ABB RobotStudio station: Station_[09.05.13]3.rsstn

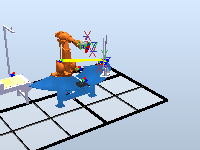
Station Station_[09.05.13] (saved by RobotStudio format 3)
Controller IRB2400_10kg_1.5m_3, task T_ROB1: task frame (RAPID world) sits at (0, 0, 226) mm in the station
Controller IRB2400_10kg_1.5m_3
  mechanical unit ROB_1: IRB2400_10_150__02, 6 joints, base frame (0, 0, -10) mm
Layout (positions relative to the parent item):
  - IRB2400_10_150__02 [mechanism, from Robots\IRB2400_10_150__02.rslib] at (0, 0, 216) mm; joint values [0, 0, 0, 0, 0, 0] (rad or m)
  - Table3_2 [part]
  - SC_RightDispenser [smart component] at (848.89, 660.39, 707) mm, rotated rx 0 ry 0 rz -142.5 deg
      signals: DI diNewPin, DO doPinInPosition2, DO doPinInPosition1
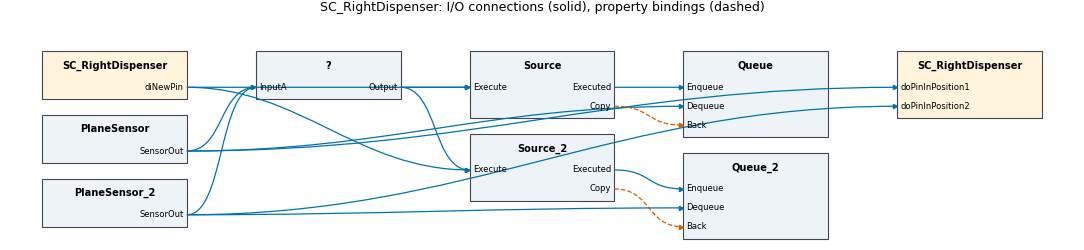
      connections:
        SC_RightDispenser.diNewPin -> Source.Execute
        Source.Executed -> Queue.Enqueue
        PlaneSensor.SensorOut -> Queue.Dequeue
        PlaneSensor.SensorOut -> SC_RightDispenser.doPinInPosition1
        PlaneSensor.SensorOut -> ?.InputA
        ?.Output -> Source.Execute
        SC_RightDispenser.diNewPin -> Source_2.Execute
        Source_2.Executed -> Queue_2.Enqueue
        PlaneSensor_2.SensorOut -> Queue_2.Dequeue
        PlaneSensor_2.SensorOut -> SC_RightDispenser.doPinInPosition2
        PlaneSensor_2.SensorOut -> ?.InputA
        ?.Output -> Source_2.Execute
        Source.Copy => Queue.Back
        Source_2.Copy => Queue_2.Back
    - Dispenser [part]
    - Source [smart component]
        properties: Source=Pin; Copy=(none); Parent=(none); Position=[-0.078 0.0985 0.189]; Orientation=[0 0 0]; Transient=false
        signals: DI Execute, DO Executed
    - Queue [smart component]
        properties: Back=(none); Front=(none); Queue={baa7ba2a-e563-400f-ae00-338ac9d6b310};{166c1fa7-f084-4893-8c68-a7378bc4935a};{0c8467ce-4cb3-4075-8f36-e6447ecc44ba};{a4931bd6-61c0-4022-957d-34420e4f6ad0};{b2f85a70-4d19-413a-b019-3afa180c1445};{512256d1-278f-462d-98f1-9ffcbd4d9afc};{849db594-4dfe-4c58-a8bd-451d21853566};{c968444c-bd1a-4f2f-bbaa-bfd3e7f50be5};{53c4b951-dfc2-4c08-b51d-efe4876241dc};{64f07cc2-7ba3-4255-a888-147bdde81c96};{5e5e12c0-75f5-4fd7-8049-5710cdd06950};{7bc2919c-0f2a-489c-9e4c-df3bff6561ed};{5aa4b278-0833-4ca9-af8d-253aa8523874};{1baac950-fc54-4ea7-852c-7f888843f6f9};{b4b16473-bd2b-40f5-a110-90fbcba822d9};{d003a69b-5307-4c56-b226-d498155ba824};{d659394f-77c7-41ee-9797-cd61472f6401};{a8294731-aa9f-4324-81a7-55ebbef1ff1c};{1eff712e-2c63-4fa8-99b0-fad1482486d3};{b15f9735-19cd-4f7a-8d4f-e540a16427f5};{02485707-3f80-4cc3-94a6-af0fe382acfb};{ec0e8ce0-b480-4ff5-b740-0a7d244ffb35};{21e78636-7eb3-4061-8dde-926c3e464303};{0772fef3-b80e-464b-9cad-322a585d167a};{d8ed8ead-e522-4938-9c7c-7997e1d5aae1};{4dfefca0-2913-4484-9455-684dfc1cbf5a};{f8c8569f-a97f-4f57-84f0-3da59c0f2755};{9fd95979-e5cf-4fa7-b177-2c560699c82c};{84f56170-3294-4345-a728-b2bfe69be833};{b3710d51-6f0f-48ac-9b0f-811ac7c7d083};{c8300349-23e3-4531-beb4-4210900096fb};{31c2e06e-432b-4cd5-8dfd-12cdd0c38bbf};{f6bc1e00-ec05-46bf-9f1a-fcc25cb6084b};{46f4262a-e9c9-45b1-8eff-bed77a1a9e5b};{07cc3b07-c3da-44db-b33b-99881492d9cc};{0c369fdb-a0e7-4beb-a0c1-abd25c6b2a43};{d9cb4cdb-12a7-4146-bf1e-65335fe6fd56};{f09a15e7-f9e4-4c16-add7-657cccb8590f}; NumberOfObjects=0
        signals: DI Enqueue, DI Dequeue, DI Clear, DI Delete, DI DeleteAll
    - LinearMover [smart component]
        properties: Object=Queue; Direction=[0 0 -0.07]; Speed=0.05; Reference=Global; ReferenceObject=(none)
        signals: DI Execute
    - PlaneSensor [smart component]
        properties: Origin=[-0.0530000000000006 0.1235 0.1195]; Axis1=[-0.03 0 0]; Axis2=[0 -0.04 0]; SensedPart=(none)
        signals: DI Active, DO SensorOut
      - _sensorPart_ [part]
    - Pin [part] at (-78, 98.5, 189) mm
    - Source_2 [smart component]
        properties: Source=Pin_2; Copy=(none); Parent=(none); Position=[-0.078 -0.0985 0.198]; Orientation=[0 0 0]; Transient=false
        signals: DI Execute, DO Executed
    - Queue_2 [smart component]
        properties: Back=(none); Front=(none); Queue={1c26a820-5f81-4fc8-b661-270a696b215b};{079caa1e-4b65-4731-ac2d-b38991013e84};{04249497-c8e4-4d2b-8d23-0d0c3b1232f2};{9b46111e-8043-4ec7-820f-f6b1f3216e0a};{190405bf-72c0-4a75-968d-0e05791ba659};{cdaa2867-23d2-4f9c-8306-ddafce1e9ac9};{a0d1b5cc-bcdc-4e7d-b91f-09bc5bc174e5};{802900b3-44c0-4e10-9d61-adfd75a0d86d};{e1828195-6a4a-4e48-b78f-f1287aff9cdc};{27d5d252-1980-452a-aff5-49173c411714};{b44ede4c-8dd3-43ce-8da4-3f1fb091dc7f};{168b000f-829e-439e-a2b5-5bc5735400ce};{aacdfd62-2178-4132-b345-2cd6db76197d};{33bd895a-7dcf-445c-8a77-0a7b01e583dc};{c1a42cbc-38c3-48e5-a615-b149ac9d8780};{fcea76f5-b349-47ef-a520-1d1e9307533b};{d936eec8-07d3-4a18-b33b-be549f4009da};{161ff837-8ce6-447d-8217-59dc5e5add53};{a4db4600-beb4-451b-b75b-f36278185638};{fac26080-080b-42e5-8e31-79509598499f};{631b6ef4-884c-4e99-a73e-a0a20b005bbd};{c6922cb5-858b-4dce-bc49-d50c5bb6ff29};{df2a1232-f236-477f-a341-c0e7247ec374};{648e1593-9b95-4c8f-9a3a-4728290fef8c};{9aba8fcf-9d7f-441d-92fe-144ce1ccaea8}; NumberOfObjects=0
        signals: DI Enqueue, DI Dequeue, DI Clear, DI Delete, DI DeleteAll
    - LinearMover_2 [smart component]
        properties: Object=Queue_2; Direction=[0 0 -0.07]; Speed=0.05; Reference=Global; ReferenceObject=(none)
        signals: DI Execute
    - PlaneSensor_2 [smart component]
        properties: Origin=[-0.053 -0.1235 0.1195]; Axis1=[-0.03 0 0]; Axis2=[0 0.04 0]; SensedPart=(none)
        signals: DI Active, DO SensorOut
      - _sensorPart_ [part]
    - Pin_2 [part] at (-78, -98.5, 189) mm
  - Pallet [part] at (1211.56, -23.95, 701.75) mm, rotated rx 0 ry -0.05 rz -179.99 deg
  - NewSmartGripper[040513] [smart component] at (940, 0, 1671) mm, rotated rx 0 ry 90 rz 0 deg
      signals: DO doPinAttached, DI diAttachPin, DO doPalletAttached, DO doGripperTouchesTable
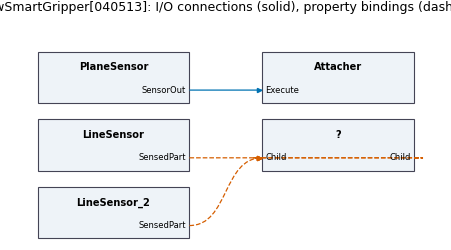
      connections:
        PlaneSensor.SensorOut -> Attacher.Execute
        LineSensor.SensedPart => ?.Child
        ?.Child => ?.Child
        LineSensor_2.SensedPart => ?.Child
        ?.Child => ?.Child
    - LineSensor [smart component, from Components\LineSensor.rslib]
        properties: Start=[0.03 0 0.1702]; End=[0.03 0 0.16]; Radius=0.002; SensedPart=(none); SensedPoint=[0 0 0]
      - _sensorPart_ [part]
    - LineSensor_2 [smart component, from Components\LineSensor.rslib]
        properties: Start=[-0.109 0.07175 0.18]; End=[-0.109 0.07175 0.1]; Radius=0.0012; SensedPart=(none); SensedPoint=[0 0 0]
      - _sensorPart_ [part]
    - LineSensor_3 [smart component, from Components\LineSensor.rslib]
        properties: Start=[-0.142 0 0.04]; End=[-0.12 0 0.04]; Radius=0.004; SensedPart=(none); SensedPoint=[0 0 0]
      - _sensorPart_ [part]
    - PoseMover [smart component, from Components\PoseMover.rslib]
        properties: Mechanism=NewGripperMech; Pose=3; Duration=0.2
    - PoseMover_2 [smart component, from Components\PoseMover.rslib]
        properties: Mechanism=NewGripperMech; Pose=2; Duration=0.2
    - NewGripperMech [mechanism] at (0, 0, 0) mm; joint values [-0.008, 0.008] (rad or m)
        TCP tTine at (-114.5, 0, 234.15) mm, rotated rx 0 ry 0 rz 180 deg
        TCP tGrip at (30, 0, 180) mm, rotated rx 0 ry -90 rz 0 deg
        links: L1, L2, L3
    - LogicGateDetachPin [smart component, from Components\LogicGate.rslib]
        properties: Operator=NOT; Delay=0
    - LogicSRLatchPalletAttached [smart component, from Components\LogicSRLatch.rslib]
    - LogicGateTouchTableANDPallet [smart component, from Components\LogicGate.rslib]
        properties: Operator=AND; Delay=0
    - PlaneSensor [smart component, from Components\PlaneSensor.rslib]
        properties: Origin=[-0.1 -0.05 0.055]; Axis1=[0.02 0 0]; Axis2=[0 0.1 0]; SensedPart=(none)
      - _sensorPart_ [part]
    - LinearMover [smart component, from Components\LinearMover.rslib]
        properties: Object=Pallet; Direction=[0 0 -1]; Speed=0.1; Reference=Object; ReferenceObject=PlaneSensor
    - Positioner [smart component, from Components\Positioner.rslib]
        properties: Object=Pallet; Position=[-0.143 -0.11 0.273]; Orientation=[0 1.5707963267949 0]; Reference=Object; ReferenceObject=PlaneSensor
    - Attacher [smart component, from Components\Attacher.rslib]
        properties: Parent=NewSmartGripper[040513]; Flange=0; Child=Pallet; Mount=false; Offset=[0 0 0]; Orientation=[0 0 0]
    - LinearMover_stop [smart component, from Components\LinearMover.rslib]
        properties: Object=Pallet; Direction=[0 0 1E-07]; Speed=1E-07; Reference=Object; ReferenceObject=PlaneSensor
  - SmartComponent_1 [smart component]
  - SC_Conveyor[190413] [smart component, from rs\SC_Conveyor[190413].rslib] at (45.5, -3634, 0) mm
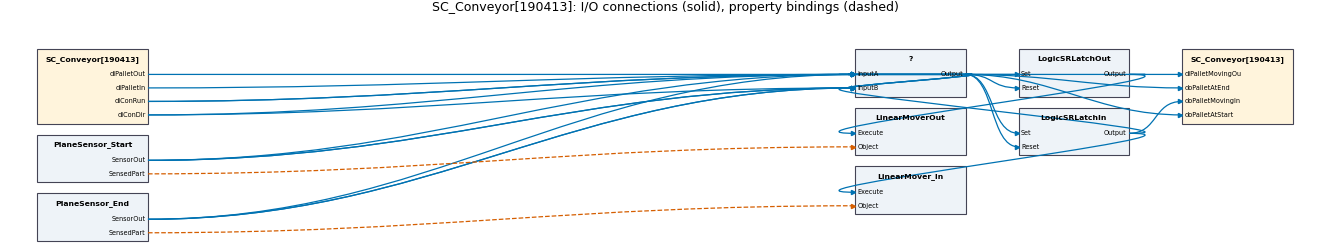
      connections:
        SC_Conveyor[190413].diPalletOut -> ?.InputA
        PlaneSensor_Start.SensorOut -> ?.InputB
        PlaneSensor_Start.SensorOut -> ?.InputA
        ?.Output -> ?.InputA
        ?.Output -> ?.InputB
        ?.Output -> LogicSRLatchOut.Set
        LogicSRLatchOut.Output -> LinearMoverOut.Execute
        LogicSRLatchOut.Output -> SC_Conveyor[190413].diPalletMovingOut
        ?.Output -> ?.InputA
        PlaneSensor_End.SensorOut -> ?.InputB
        ?.Output -> LogicSRLatchOut.Reset
        ?.Output -> SC_Conveyor[190413].doPalletAtEnd
        SC_Conveyor[190413].diPalletIn -> ?.InputA
        PlaneSensor_End.SensorOut -> ?.InputB
        PlaneSensor_End.SensorOut -> ?.InputA
        ?.Output -> ?.InputA
        ?.Output -> ?.InputB
        ?.Output -> LogicSRLatchIn.Set
        LogicSRLatchIn.Output -> LinearMover_In.Execute
        LogicSRLatchIn.Output -> SC_Conveyor[190413].doPalletMovingIn
        ?.Output -> ?.InputA
        PlaneSensor_Start.SensorOut -> ?.InputB
        ?.Output -> LogicSRLatchIn.Reset
        ?.Output -> SC_Conveyor[190413].doPalletAtStart
        LogicSRLatchOut.Output -> ?.InputA
        LogicSRLatchIn.Output -> ?.InputB
        ?.Output -> ?.InputA
        SC_Conveyor[190413].diConRun -> ?.InputA
        SC_Conveyor[190413].diConDir -> ?.InputA
        ?.Output -> ?.InputB
        ?.Output -> ?.InputA
        SC_Conveyor[190413].diConRun -> ?.InputA
        SC_Conveyor[190413].diConDir -> ?.InputB
        ?.Output -> ?.InputA
        PlaneSensor_Start.SensedPart => LinearMoverOut.Object
        PlaneSensor_End.SensedPart => LinearMover_In.Object
    - Conveyor3 [part, from rs\SC_Conveyor[190413].rslib] at (0, 0, 606) mm
    - PlaneSensor_Start [smart component, from Libraries\SC_RightDispenser[080513].rslib]
        properties: Origin=[-0.05 0.4 0.62]; Axis1=[-0.5 0 0]; Axis2=[0 2.1 0]; SensedPart=(none)
      - _sensorPart_ [part, from rs\SC_Conveyor[190413].rslib]
    - PlaneSensor_End [smart component, from Libraries\SC_RightDispenser[080513].rslib]
        properties: Origin=[-0.05 0 0.62]; Axis1=[-0.5 0 0]; Axis2=[0 2.2 0]; SensedPart=(none)
      - _sensorPart_ [part, from rs\SC_Conveyor[190413].rslib]
    - LinearMoverOut [smart component, from Libraries\SC_RightDispenser[080513].rslib]
        properties: Object=(none); Direction=[0 -1 0]; Speed=0.6; Reference=Global; ReferenceObject=(none)
    - LinearMover_In [smart component, from Libraries\SC_RightDispenser[080513].rslib]
        properties: Object=(none); Direction=[0 1 0]; Speed=0.6; Reference=Global; ReferenceObject=(none)
    - LogicSRLatchOut [smart component, from rs\SC_Conveyor[190413].rslib]
    - LogicSRLatchIn [smart component, from rs\SC_Conveyor[190413].rslib]
  - Frame_1 [frame] at (710.04, 677.11, 1017.54) mm, rotated rx -135.34 ry 89.95 rz -97.28 deg
Attachment: NewSmartGripper[040513] is attached to IRB2400_10_150__02 / Link6
EventTableEntry 5: Group=, Trigger=Grip 6, Actions=[diGRIP 7], Comment=, ActivationMode=2, Cyclic=false
EventTableTriggerIO 6: IOValue=[1], IRC5Controller=? -1, Operator=0, SignalSource=IRB2400_10kg_1.5m_3 486
EventTableActionIO 7: IOValue=[0], IRC5Controller=? -1, SignalTarget=Station_[09.05.13] 1
EventTableEntry 8: Group=, Trigger=Grip 9, Actions=[diGRIP 10], Comment=, ActivationMode=2, Cyclic=false
EventTableTriggerIO 9: IOValue=[0], IRC5Controller=? -1, Operator=0, SignalSource=IRB2400_10kg_1.5m_3 486
EventTableActionIO 10: IOValue=[1], IRC5Controller=? -1, SignalTarget=Station_[09.05.13] 1
EventTableTriggerIO 1726: IOValue=[1], IRC5Controller=? -1, Operator=0, SignalSource=IRB2400_10kg_1.5m_3 486
EventTableTriggerIO 1727: IOValue=[0], IRC5Controller=? -1, Operator=0, SignalSource=IRB2400_10kg_1.5m_3 486
EventTableEntry 1775: Group=, Trigger=ConRun 1776, Actions=[diStationConRun 1777], Comment=, ActivationMode=2, Cyclic=false
EventTableTriggerIO 1776: IOValue=[1], IRC5Controller=? -1, Operator=0, SignalSource=IRB2400_10kg_1.5m_3 486
EventTableActionIO 1777: IOValue=[1], IRC5Controller=? -1, SignalTarget=Station_[09.05.13] 1
EventTableEntry 1778: Group=, Trigger=ConDir 1779, Actions=[diStationConDir 1780], Comment=, ActivationMode=2, Cyclic=false
EventTableTriggerIO 1779: IOValue=[1], IRC5Controller=? -1, Operator=0, SignalSource=IRB2400_10kg_1.5m_3 486
EventTableActionIO 1780: IOValue=[1], IRC5Controller=? -1, SignalTarget=Station_[09.05.13] 1
EventTableEntry 1781: Group=, Trigger=ConRun 1782, Actions=[diStationConRun 1783], Comment=, ActivationMode=2, Cyclic=false
EventTableTriggerIO 1782: IOValue=[0], IRC5Controller=? -1, Operator=0, SignalSource=IRB2400_10kg_1.5m_3 486
EventTableActionIO 1783: IOValue=[0], IRC5Controller=? -1, SignalTarget=Station_[09.05.13] 1
EventTableEntry 1784: Group=, Trigger=ConDir 1785, Actions=[diStationConDir 1786], Comment=, ActivationMode=2, Cyclic=false
EventTableTriggerIO 1785: IOValue=[0], IRC5Controller=? -1, Operator=0, SignalSource=IRB2400_10kg_1.5m_3 486
EventTableActionIO 1786: IOValue=[0], IRC5Controller=? -1, SignalTarget=Station_[09.05.13] 1
Collision set CollisionSet_1:  against , near miss 0 m
Station signals: DI diRunConOUT, DI diRunConIN, DI diGRIP, DI diNewPinINDISP, DI diStationConRun, DI diStationConDir
Station logic (signal -> signal, property => property):
  Station_[09.05.13].diGRIP -> NewSmartGripper[040513].diAttachPin
  Station_[09.05.13].diNewPinINDISP -> SC_RightDispenser.diNewPin
  Station_[09.05.13].diStationConRun -> ?.diConRun
  Station_[09.05.13].diStationConDir -> ?.diConDir
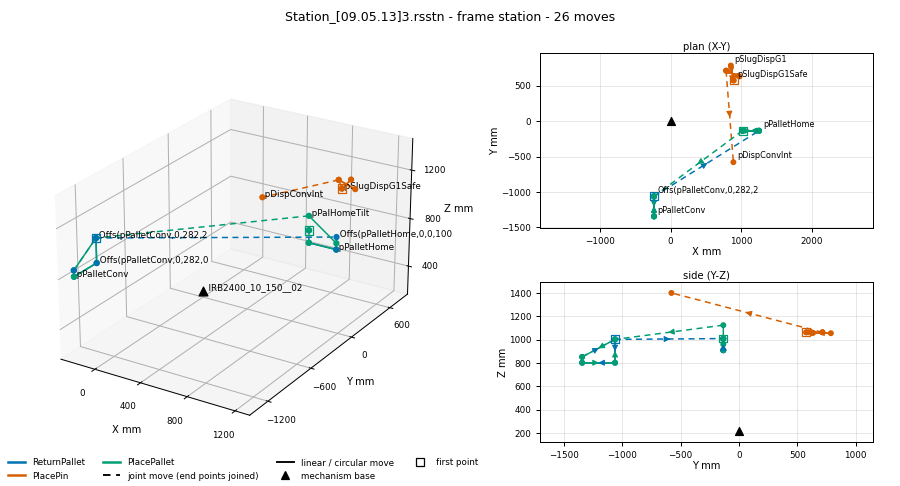
[picture p0: tool path of Station_[09.05.13]3.rsstn in frame station, 26 of 38 moves have a stored position in this frame; points joined in program order, loops and branches not executed]
Targets, tools, work objects and paths stored in the station, written as RAPID:
! task T_ROB1
MODULE MW
  PERS tooldata tGrip:=[TRUE,[[30,0,180],[1,0,0,0]],[1.5,[0,0,80],[1,0,0,0],0,0,0]];
  PERS tooldata tTine:=[TRUE,[[-114.5,0,234.15],[1,0,0,0]],[1.5,[0,0,80],[1,0,0,0],0.04,0.04,0.04]];
  CONST robtarget pPalletConv:=[[-234.56,-1344.02,576.85],[0.500039998,0.499942998,-0.500039998,0.499976998],[-2,-1,-2,0],[9E9,9E9,9E9,9E9,9E9,9E9]];
  CONST robtarget pPalletHome:=[[1250.04,-133.95,684.28],[0.000048,-0.707407715,-0.000048,-0.706805716],[-1,-1,-2,0],[9E9,9E9,9E9,9E9,9E9,9E9]];
  CONST jointtarget jtCalibPos:=[[0,0,0,0,0,0],[9E9,9E9,9E9,9E9,9E9,9E9]];
  CONST robtarget pSlugDispG1Safe:=[[890.6,577.3,837.9],[0.678140503,-0.200710149,0.678000503,0.200390149],[0,0,-1,0],[9E9,9E9,9E9,9E9,9E9,9E9]];
  CONST robtarget pSlugDispG1:=[[851.75,788.07,830.08],[0.668320736,-0.230855909,0.668581736,0.230328909],[0,0,-1,0],[9E9,9E9,9E9,9E9,9E9,9E9]];
  CONST robtarget pSlugDispG2Safe:=[[784.1,715.6,837.7],[0.658308518,-0.269043481,0.654098463,0.257683334],[0,-1,0,0],[9E9,9E9,9E9,9E9,9E9,9E9]];
  CONST robtarget pSlugDispG2:=[[974.96,633.73,831.83],[0.668405716,-0.230831902,0.668514716,0.230300902],[0,-1,0,0],[9E9,9E9,9E9,9E9,9E9,9E9]];
  CONST robtarget pDispConvInt:=[[887.7,-578.4,1175.2],[0.654679605,0.26514984,0.656439604,-0.26490984],[-1,-1,0,0],[9E9,9E9,9E9,9E9,9E9,9E9]];
  CONST robtarget pPalHomeTilt:=[[1015.987042359,-133.981901811,898.978895592],[0.000045049,-0.665857682,-0.00005045,-0.746078778],[-1,-1,-2,0],[9E9,9E9,9E9,9E9,9E9,9E9]];
  PROC main()
  ENDPROC
  PROC ReturnPallet()
    MoveJ Offs(pPalletConv,0,282,200),v1000,fine,tTine;
    MoveL Offs(pPalletConv,0,282,0),v200,fine,tTine;
    MoveL pPalletConv,v200,fine,tTine;
    MoveL Offs(pPalletConv, 0,0,50),v200,fine,tTine;
    MoveJ Offs(pPalletConv,0,282,200),v1000,fine,tTine;
    MoveJ Offs(pPalletHome,0,0,100),v1000,fine,tTine;
    MoveL pPalletHome,v200,fine,tTine;
    MoveL Offs(pPalletHome,-232,0,0),v500,fine,tTine;
    MoveJ Offs(pPalletHome,-232,0,100),v1000,fine,tTine;
    MoveAbsJ jtCalibPos,v1000,fine,tTine;
  ENDPROC
  PROC RemovePin()
    MoveJ Offs(pSlugPallConvCD,0,0,100),v1000,fine,tGrip;
    Set Grip;
    MoveL Offs(pSlugPallH1G, xoffset, yoffset, 50),v200,fine,tGrip;
    MoveL Offs(pSlugPallH1G, xoffset, yoffset, 0),v200,fine,tGrip;
    Reset Grip;
    WaitTime 1;
    MoveL Offs(pSlugPallH1G, xoffset, yoffset, 200),v200,fine,tGrip;
    MoveAbsJ jtCalibPos,v1000,fine,tTine;
    Reset Grip;
  ENDPROC
  PROC PlacePin()
    MoveJ pSlugDispG1Safe,v500,fine,tGrip;
    MoveL pSlugDispG1,v200,fine,tGrip;
    Set Grip;
    WaitTime 1;
    MoveL pSlugDispG1Safe,v200,fine,tGrip;
    MoveJ pSlugDispG2Safe,v1000,fine,tGrip;
    MoveL pSlugDispG2,v200,fine,tGrip;
    Set Grip;
    WaitTime 1;
    MoveL pSlugDispG2Safe,v200,fine,tGrip;
    MoveJ pDispConvInt,v1000,fine,tGrip;
    MoveJ Offs(pSlugPallConvCD,0,0,200),v1000,fine,tGrip;
    MoveL Offs(pSlugPallH1D, xoffset, yoffset, 50),v200,fine,tGrip;
    MoveL Offs(pSlugPallH1D, xoffset, yoffset, 0),v200,fine,tGrip;
    Reset Grip;
    WaitTime 1;
    MoveL Offs(pSlugPallH1D, xoffset, yoffset, 100),v200,fine,tGrip;
    MoveAbsJ jtCalibPos,v1000,fine,tTine;
  ENDPROC
  PROC PlacePallet()
    MoveJ Offs(pPalletHome,-232,0,100),v1000,fine,tTine;
    MoveJ Offs(pPalletHome,-232,0,0),v500,fine,tTine;
    MoveL pPalletHome,v200,fine,tTine;
    MoveL Offs(pPalletHome,0,0,50),v200,fine,tTine;
    MoveL pPalHomeTilt,v200,fine,tTine;
    MoveJ Offs(pPalletConv,0,282,200),v1000,fine,tTine;
    MoveL Offs(pPalletConv,0,0,50),v500,fine,tTine;
    MoveL pPalletConv,v200,fine,tTine;
    MoveL Offs(pPalletConv,0,282,0),v200,fine,tTine;
    MoveL Offs(pPalletConv,0,282,200),v500,fine,tTine;
    MoveAbsJ jtCalibPos,v1000,fine,tTine;
  ENDPROC
ENDMODULE

! task T_ROB1
MODULE CalibData
  PERS tooldata Tooldata_1:=[TRUE,[[20,0,175.76],[0.707106781,0,-0.707106781,0]],[1,[0,0,1],[1,0,0,0],0,0,0]];
  PERS tooldata Tooldata_2:=[TRUE,[[-83.5,0,233],[0,0.707106781,0,0.707106781]],[1,[0,0,1],[1,0,0,0],0,0,0]];
  PERS tooldata My_Mechanism_1:=[TRUE,[[20,0,175.76],[0.707106781,0,-0.707106781,0]],[1,[0,0,1],[1,0,0,0],0,0,0]];
  PERS tooldata My_Mechanism_2:=[TRUE,[[-83.5,0,233],[0,0.707106781,0,0.707106781]],[1,[0,0,1],[1,0,0,0],0,0,0]];
ENDMODULE

